{attribute 'linkalways'} 
{attribute 'no_explicit_call' := 'This FB is a CLASS and must be accessed using methods or properties'}
{attribute 'enable_dynamic_creation'}
FUNCTION_BLOCK Node_F_VN_ReadBarcodeExp EXTENDS VisionNode
VAR
    ipSrcImage : _ITcVnImage;
    ipDecodedData : _ITcVnContainer;
	ipContours : _ITcVnContainer;
    eBarcodeType : _ETcVnBarcodeType(ETcVnBarcodeType.TCVN_BT_ANY);
	nCodeNumber : _DINT(1);
	eSearchDirection : _ETcVnBarcodeSearchDirection(ETcVnBarcodeSearchDirection.TCVN_BSD_ANY);
    hrPrev : _HRESULT(S_OK);
	hresult : _HRESULT(S_OK);
END_VAR

METHOD PUBLIC  Clone : I_Node
VAR
	pNode : POINTER TO Node_F_VN_ReadBarcodeExp;
END_VAR
pNode := __NEW(Node_F_VN_ReadBarcodeExp);
Clone := pNode^;
END_METHOD

METHOD FB_init : BOOL
VAR_INPUT
	bInitRetains : BOOL; // if TRUE, the retain variables are initialized (warm start / cold start)
	bInCopyCode : BOOL;  // if TRUE, the instance afterwards gets moved into the copy code (online change)
END_VAR
AddInput('ipSrcImage', ipSrcImage);
AddParameter('eBarcodeType', eBarcodeType);
AddParameter('nCodeNumber', nCodeNumber);
AddParameter('eSearchDirection', eSearchDirection);
AddInput('hrPrev', hrPrev);
AddOutput('ipDecodedData', ipDecodedData);
AddOutput('ipContours', ipContours);
AddOutput('hresult',hresult);
END_METHOD

METHOD PROTECTED OnExecute
hresult.Value := F_VN_ReadBarcodeExp(
	ipSrcImage := ipSrcImage.Value,
    ipDecodedData := ipDecodedData.Value,
	ipContours := ipContours.Value,
    eBarcodeType := eBarcodeType.Value,
	nCodeNumber := nCodeNumber.Value,
	eSearchDirection := eSearchDirection.Value,
	hrPrev:= hrPrev.Value);
END_METHOD

METHOD PUBLIC PreExecutionCheck
VAR_INPUT
	Check : I_PreExecutionChecks;
END_VAR
Check.IsTrue(ipSrcImage.IsValid, 'ipSrcImage must contain an image');
Check.IsTrue((ipSrcImage.HasChannelCount(1) OR ipSrcImage.HasChannelCount(3)), 'ipSrcImage must have 1 or 3 channels');
Check.IsTrue(ipSrcImage.IsPixelDepth(8), 'ipSrcImage must have 8 bit pixel depth');
Check.IsTrue((nCodeNumber.Value = 1), 'nCodeNumber, currently only 1 supported');
END_METHOD

END_FUNCTION_BLOCK

(* stored: Version 1.1.0.1, ProductVersion 3.1.4026.13
   POU Node_F_VN_ReadBarcodeExp: Id {aa70d419-c39e-04cb-0580-1c143e427c02}, SpecialFunc None
   Folder Constructor: Id {72546c85-481b-07ca-17d4-b9440ce9cbfa}
   Method Clone: Id {5d60b9ac-6882-017c-0942-a247fff3c59e}
   Method FB_init: Id {c7dde6ff-574c-009f-086c-2bf3584f97da}
   Method OnExecute: Id {2b1ecbf7-6dc5-03c9-2c3b-26f3565b617e}
   Method PreExecutionCheck: Id {709d848d-f38b-0430-2f9e-dd3634ceb475} *)
